(* IEC 61131-3 sources: volt/packages/volt-lsp-iec/test-corpus/awa-palletizer/Device/Plc Logic/Application/Library Manager/(unresolved)/alarm manager interfaces, 21 files *)

(* ---- ALARM_ID.dut ---- *)
TYPE ALARM_ID : UINT;
END_TYPE

(* ---- STRUCTFILTERINGNAME.dut ---- *)
TYPE STRUCTFILTERINGNAME :
STRUCT
	SREMOTEDEVICE : STRING;
	SNAME : STRING;
END_STRUCT
END_TYPE

(* ---- TIMESTAMP.dut ---- *)
TYPE TIMESTAMP : LINT;
END_TYPE

(* ---- ALARMSERVICECONSTANTS.gvl ---- *)
VAR_GLOBAL
	SG_ALARMMANAGER : UINT := 16#18;
	COMMAND_GET_ALARM_COUNT : UINT := 16#81;
	COMMAND_GET_ALARMS : UINT := 16#82;
	COMMAND_GET_ALARMS2 : UINT := 16#83;
	COMMAND_GET_MIN_MAX_TIMESTAMPS : UINT := 16#84;
	COMMAND_GET_ALARMS3 : UINT := 16#85;
	COMMAND_GET_ACTIVE_ALARMS : UINT := 16#86;
	COMMAND_GET_ALARM_CONFIGURATION : UINT := 16#87;
	COMMAND_ACKNOWLEDGE : UINT := 16#89;
	COMMAND_CHANNEL_TEST : UINT := 16#8A;
	COMMAND_SET_ALARM_RECORD : UINT := 16#8B;
	COMMAND_RES_ALARM_RECORD : UINT := 16#8C;
	COMMAND_GET_ACTIVE_ALARMS2 : UINT := 16#8D;
	COMMAND_GET_ALARM_CONFIGURATION2 : UINT := 16#8E;
	COMMAND_GET_CLASS_CONFIGURATION : UINT := 16#8F;
	COMMAND_GET_HIST_CONFIGURATION : UINT := 16#90;
	COMMAND_GET_HIST_ALARMS : UINT := 16#91;
	COMMAND_GET_HIST_ACTIVE_ALARMS : UINT := 16#92;
	TAG_APPLICATION_NAME : UINT := 16#1;
	TAG_ALARMGROUP_IDS : UINT := 16#2;
	TAG_ALARMCLASS_IDS : UINT := 16#3;
	TAG_PRIORITY : UINT := 16#4;
	TAG_ROW_SPECIFICATION : UINT := 16#5;
	TAG_ROW_ID : UINT := 16#6;
	TAG_GET_ALARMS3_PARAMETER : UINT := 16#7;
	TAG_GET_ALARMS3_GLOBAL_PARAMETER : UINT := 16#8;
	TAG_COUNT_SUBELEMENTS : UINT := 16#9;
	TAG_ALARMGROUP : UINT := 16#A;
	TAG_ALARMCLASS : UINT := 16#B;
	TAG_ALARM_FILTER_LATCH : UINT := 16#C;
	TAG_CHANNEL_TEST : UINT := 16#D;
	TAG_ID : UINT := 16#E;
	TAG_ALARM_FILTER_TR : UINT := 16#F;
	TAG_ALARMGROUPS : UINT := 16#86;
	TAG_ALARMCLASSES : UINT := 16#87;
	TAG_ACKNOWLEDGE : UINT := 16#2C;
	TAG_GET_ALARM_COUNT_REPLY : UINT := 16#1;
	TAG_ALARM_RECORD : UINT := 16#2;
	TAG_HIST_ALARM_DB_STATUS : UINT := 16#1;
	TAG_GET_ALARMS_REPLY : UINT := 16#82;
	TAG_GET_ALARMS2_REPLY : UINT := 16#83;
	TAG_HIST_ALARM : UINT := 16#82;
	TAG_HIST_ALARM_ROW : UINT := 16#1;
	TAG_HIST_ALARM_LATCH_VARIABLE : UINT := 16#2;
	TAG_HIST_ALARM_CLOSE : UINT := 16#3;
	TAG_HIST_ALARM_DBDATA : UINT := 16#4;
	SUBT_GET_ALARMS_REPLY_ERROR : UINT := 16#1;
	SUBT_GET_ALARMS_REPLY_ROWS : UINT := 16#2;
	SUBT_GET_ALARMS_REPLY_ROW_ID : UINT := 16#3;
	SUBT_GET_ALARMS2_ALARM : UINT := 16#84;
	SUBT_GET_ALARMS2_ALARM_CONSTANT_VALUES : UINT := 16#21;
	SUBT_GET_ALARMS2_ALARM_LATCH_VARIABLE : UINT := 16#22;
	SUBT_GET_ALARMS2_ALARM_STRING_LATCH_VARIABLE : UINT := 16#32;
	SUBT_GET_ALARMS2_ALARM_OFFSET : UINT := 16#33;
	SUBT_GET_MIN_MAX_TIMESTAMPS : UINT := 16#23;
	SUBT_GET_ALARMS3_RESULT : UINT := 16#24;
	SUBT_GET_ACTIVE_ALARMS_ALARMID : UINT := 16#25;
	SUBT_GET_ACTIVE_ALARMS_ALARMGROUPNAME : UINT := 16#26;
	SUBT_GET_ACTIVE_ALARMS_ALARMCLASSNAME : UINT := 16#27;
	SUBT_GET_ACTIVE_ALARMS_TEXTLISTNAME : UINT := 16#28;
	SUBT_GET_ALARMCONF_ALARMGROUP : UINT := 16#85;
	SUBT_GET_ALARMCONF_ALARMGROUP_DESCRIPTION : UINT := 16#29;
	SUBT_GET_ALARMCONF_ALARM_DESCRIPTION : UINT := 16#2A;
	SUBT_GET_ALARMCONF_ALARMCLASS : UINT := 16#86;
	SUBT_GET_ALARMCONF_ALARMCLASS_DESCRIPTION : UINT := 16#2B;
	SUBT_GET_ALARMCONF_ALARMSTORAGE : UINT := 16#4;
	SUBT_GET_ALARMCONF_DISPLAY_OPTIONS : UINT := 16#88;
	SUBT_GET_ALARMCONF_ALARM_STATE : UINT := 16#2D;
	SUBT_GET_ALARMCONF_FONT : UINT := 16#2E;
	SUBT_GET_ALARMCONF_BG_COLOR : UINT := 16#2F;
	SUBT_GET_ALARMCONF_BITMAP : UINT := 16#30;
	SUBT_GET_CURRENTVALUES_ALARM : UINT := 16#2A;
END_VAR

(* ---- SHERRORS.gvl ---- *)
VAR_GLOBAL
	ERR_OK : UDINT := 0;
	ERR_NOTCREATED : UDINT := 16#1000;
	ERR_NOMORETAGS : UDINT := 16#1040;
	ERR_NOCONTAINERTAG : UDINT := 16#1041;
	ERR_NODATATAG : UDINT := 16#1042;
	ERR_ENDOFTAG : UDINT := 16#1043;
	ERR_READONWRONGTAG : UDINT := 16#1044;
	ERR_MANDATORY_PARAMETER_MISSING : UDINT := 16#1045;
	ERR_UNDEF : UDINT := 16#1046;
	ERR_NOT_FOUND : UDINT := 16#1047;
	ERR_REC_NOT_GENERATED : UDINT := 16#1048;
END_VAR

(* ---- IALARMFILTERCRITERIA.itf ---- *)
INTERFACE IALARMFILTERCRITERIA
END_INTERFACE

METHOD AREALLALARMCLASSESSELECTED : BOOL
END_METHOD

METHOD AREALLALARMGROUPSSELECTED : BOOL
END_METHOD

METHOD GETALARMCLASSES : POINTER TO ARRAY [0..0] OF UDINT
END_METHOD

METHOD GETALARMGROUPS : POINTER TO ARRAY [0..0] OF UDINT
END_METHOD

METHOD GETCOUNTALARMCLASSES : INT
END_METHOD

METHOD GETCOUNTALARMGROUPS : INT
END_METHOD

METHOD GETPRIORITYFROM : USINT
END_METHOD

METHOD GETPRIORITYTO : USINT
END_METHOD

(* ---- IALARMFILTERCRITERIA2.itf ---- *)
INTERFACE IALARMFILTERCRITERIA2
END_INTERFACE

METHOD GETFILTERLATCHCONTENT : INT
END_METHOD

METHOD GETFILTERLATCHTYPEDLITERALTYPE : INT
END_METHOD

METHOD GETFILTERLATCHVALUELI : LINT
END_METHOD

METHOD GETFILTERLATCHVALUELREAL : LREAL
END_METHOD

METHOD GETFILTERLATCHVALUEREAL : REAL
END_METHOD

METHOD GETFILTERLATCHVALUEWSTRING : WSTRING
END_METHOD

METHOD ISFILTERLATCHAVAILABLE : BOOL
END_METHOD

(* ---- IALARMFILTERCRITERIA3.itf ---- *)
INTERFACE IALARMFILTERCRITERIA3
END_INTERFACE

METHOD GETALARMCLASSES3
VAR_OUTPUT
	PASTRUCTFILTERING : POINTER TO ARRAY [0..0] OF StructFilteringName;
	ICOUNT : INT;
END_VAR
END_METHOD

METHOD GETALARMGROUPS3
VAR_OUTPUT
	PASTRUCTFILTERING : POINTER TO ARRAY [0..0] OF StructFilteringName;
	ICOUNT : INT;
END_VAR
END_METHOD

(* ---- IALARMFILTERCRITERIA4.itf ---- *)
INTERFACE IALARMFILTERCRITERIA4
END_INTERFACE

METHOD GETFILTERTIMERANGEFROMVALUELI : LINT
END_METHOD

METHOD GETFILTERTIMERANGETOVALUELI : LINT
END_METHOD

METHOD GETFILTERTIMERANGETYPE : INT
END_METHOD

METHOD ISFILTERTIMERANGEAVAILABLE : BOOL
END_METHOD

(* ---- IALARMHANDLERBASE.itf ---- *)
INTERFACE IALARMHANDLERBASE
END_INTERFACE

METHOD GETALARMIDANDALARMGROUPNAME : BOOL
VAR_INPUT
	UDIALARMGROUPID : UDINT;
	UDIALARMID : UDINT;
END_VAR
VAR_OUTPUT
	SALARMGROUPNAME : STRING;
	UIALARMID : ALARM_ID;
END_VAR
END_METHOD

(* ---- IALARMMETAOBJECTSTUB3GETTER.itf ---- *)
INTERFACE IALARMMETAOBJECTSTUB3GETTER
END_INTERFACE

METHOD GETALARMGROUP : STRING
END_METHOD

METHOD GETID : ALARM_ID
END_METHOD

METHOD GETLATCHVAR1VALUE : ITypedValue
END_METHOD

METHOD GETLATCHVAR2VALUE : ITypedValue
END_METHOD

METHOD GETSTATE : INT
END_METHOD

METHOD GETTIMESTAMPACKNOWLEDGE : Timestamp
END_METHOD

METHOD GETTIMESTAMPACTIVE : Timestamp
END_METHOD

METHOD GETTIMESTAMPINACTIVE : Timestamp
END_METHOD

METHOD GETTIMESTAMPLAST : Timestamp
END_METHOD

METHOD GETTRIGGERVALUE : ITypedValue
END_METHOD

(* ---- IALARMMETAOBJECTSTUB3SETTER.itf ---- *)
INTERFACE IALARMMETAOBJECTSTUB3SETTER
END_INTERFACE

METHOD SETALARMGROUP
VAR_INPUT
	SALARMGROUP : STRING;
END_VAR
END_METHOD

METHOD SETID
VAR_INPUT
	UIID : ALARM_ID;
END_VAR
END_METHOD

METHOD SETLATCHVAR1VALUE
VAR_INPUT
	ITFTYPEDVALUELATCHVAR1 : ITypedValue;
END_VAR
END_METHOD

METHOD SETLATCHVAR2VALUE
VAR_INPUT
	ITFTYPEDVALUELATCHVAR2 : ITypedValue;
END_VAR
END_METHOD

METHOD SETSTATE
VAR_INPUT
	ISTATE : INT;
END_VAR
END_METHOD

METHOD SETTIMESTAMPACKNOWLEDGE
VAR_INPUT
	LITIMESTAMPACKNOWLEDGE : Timestamp;
END_VAR
END_METHOD

METHOD SETTIMESTAMPACTIVE
VAR_INPUT
	LITIMESTAMPACTIVE : Timestamp;
END_VAR
END_METHOD

METHOD SETTIMESTAMPINACTIVE
VAR_INPUT
	LITIMESTAMPINACTIVE : Timestamp;
END_VAR
END_METHOD

METHOD SETTIMESTAMPLAST
VAR_INPUT
	LITIMESTAMPLAST : Timestamp;
END_VAR
END_METHOD

METHOD SETTRIGGERVALUE
VAR_INPUT
	ITFTYPEDVALUETRIGGER : ITypedValue;
END_VAR
END_METHOD

(* ---- IALARMMETAOBJECTSTUB3SETTER2.itf ---- *)
INTERFACE IALARMMETAOBJECTSTUB3SETTER2
END_INTERFACE

METHOD GETCURRENTVALUE2 : ITypedValue2
END_METHOD

METHOD GETLATCHVAR1VALUE2 : ITypedValue2
END_METHOD

METHOD GETLATCHVAR2VALUE2 : ITypedValue2
END_METHOD

METHOD GETTRIGGERVALUE2 : ITypedValue2
END_METHOD

(* ---- IALARMMETAOBJECTSTUBSERVICE.itf ---- *)
INTERFACE IALARMMETAOBJECTSTUBSERVICE
END_INTERFACE

METHOD GETACKNOWLEDGE : BOOL
END_METHOD

METHOD GETACKNOWLEDGEMULTIPLE : BOOL
END_METHOD

METHOD GETALARMCLASS : STRING
END_METHOD

METHOD GETPRIORITY : BYTE
END_METHOD

METHOD GETSTRINGID : STRING
END_METHOD

METHOD GETTESTLISTNAME : STRING
END_METHOD

METHOD RESETACKNOWLEDGE
END_METHOD

METHOD SETALARMCLASS
VAR_INPUT
	SALARMCLASS : STRING;
END_VAR
END_METHOD

METHOD SETCURRENTVALUE
VAR_INPUT
	ITFTYPEDVALUECURRENT : ITypedValue;
END_VAR
END_METHOD

METHOD SETPRIORITY
VAR_INPUT
	BYPRIORITY : BYTE;
END_VAR
END_METHOD

METHOD SETSTRINGID
VAR_INPUT
	SID : STRING;
END_VAR
END_METHOD

METHOD SETTESTLISTNAME
VAR_INPUT
	STESTLISTNAME : STRING;
END_VAR
END_METHOD

(* ---- IALARMMETAOBJECTSTUBSERVICE2.itf ---- *)
INTERFACE IALARMMETAOBJECTSTUBSERVICE2
END_INTERFACE

METHOD SETACKNOWLEDGE2
VAR_INPUT
	BACKNOWLEDGEMULTIPLE : BOOL;
END_VAR
END_METHOD

(* ---- IGETALARMSREQUESTPARAMETER.itf ---- *)
INTERFACE IGETALARMSREQUESTPARAMETER
END_INTERFACE

METHOD GETALARMFILTERCRITERIA : IAlarmFilterCriteria
END_METHOD

METHOD GETMAXROWS : INT
END_METHOD

METHOD GETROWID : DINT
END_METHOD

METHOD GETROWSTOSKIP : INT
END_METHOD

METHOD ISROWIDVALID : BOOL
END_METHOD

(* ---- IGETALARMSREQUESTRESULT.itf ---- *)
INTERFACE IGETALARMSREQUESTRESULT
END_INTERFACE

METHOD GETALARMHANDLERBASE : IAlarmHandlerBase
END_METHOD

METHOD GETEFFECTIVERESULTARRAYSIZE : INT
END_METHOD

METHOD GETRESULTARRAY : POINTER TO ARRAY [0..0] OF IAlarmMetaObjectStub3Setter2
END_METHOD

METHOD SETCOUNTALARMS
VAR_INPUT
	ICOUNTALARMS : INT;
END_VAR
END_METHOD

METHOD SETROWID
VAR_INPUT
	DIROWID : DINT;
END_VAR
END_METHOD

METHOD SETROWIDVALID
VAR_INPUT
	XROWIDVALID : BOOL;
END_VAR
END_METHOD

(* ---- IGETCOUNTREQUESTPARAMETER.itf ---- *)
INTERFACE IGETCOUNTREQUESTPARAMETER
END_INTERFACE

METHOD GETALARMFILTERCRITERIA : IAlarmFilterCriteria
END_METHOD

(* ---- IGETCOUNTREQUESTRESULT.itf ---- *)
INTERFACE IGETCOUNTREQUESTRESULT
END_INTERFACE

METHOD SETCOUNTROWS
VAR_INPUT
	DICOUNTROWS : DINT;
END_VAR
END_METHOD

(* ---- ITYPEDVALUE.itf ---- *)
INTERFACE ITYPEDVALUE
END_INTERFACE

METHOD GETSIZE : INT
END_METHOD

METHOD GETTYPE : __SYSTEM.TYPE_CLASS
END_METHOD

METHOD GETVALUE : POINTER TO BYTE
END_METHOD

METHOD SETTYPE
VAR_INPUT
	TYPETOSET : __SYSTEM.TYPE_CLASS;
END_VAR
END_METHOD

METHOD SETVALUE
VAR_INPUT
	LIVALUE : LINT;
END_VAR
END_METHOD

(* ---- ITYPEDVALUE2.itf ---- *)
INTERFACE ITYPEDVALUE2
END_INTERFACE

METHOD SETRAWVALUE
VAR_INPUT
	PABYVALUE : POINTER TO ARRAY [0..7] OF BYTE;
	ETYPETOSET : __SYSTEM.TYPE_CLASS;
END_VAR
END_METHOD
